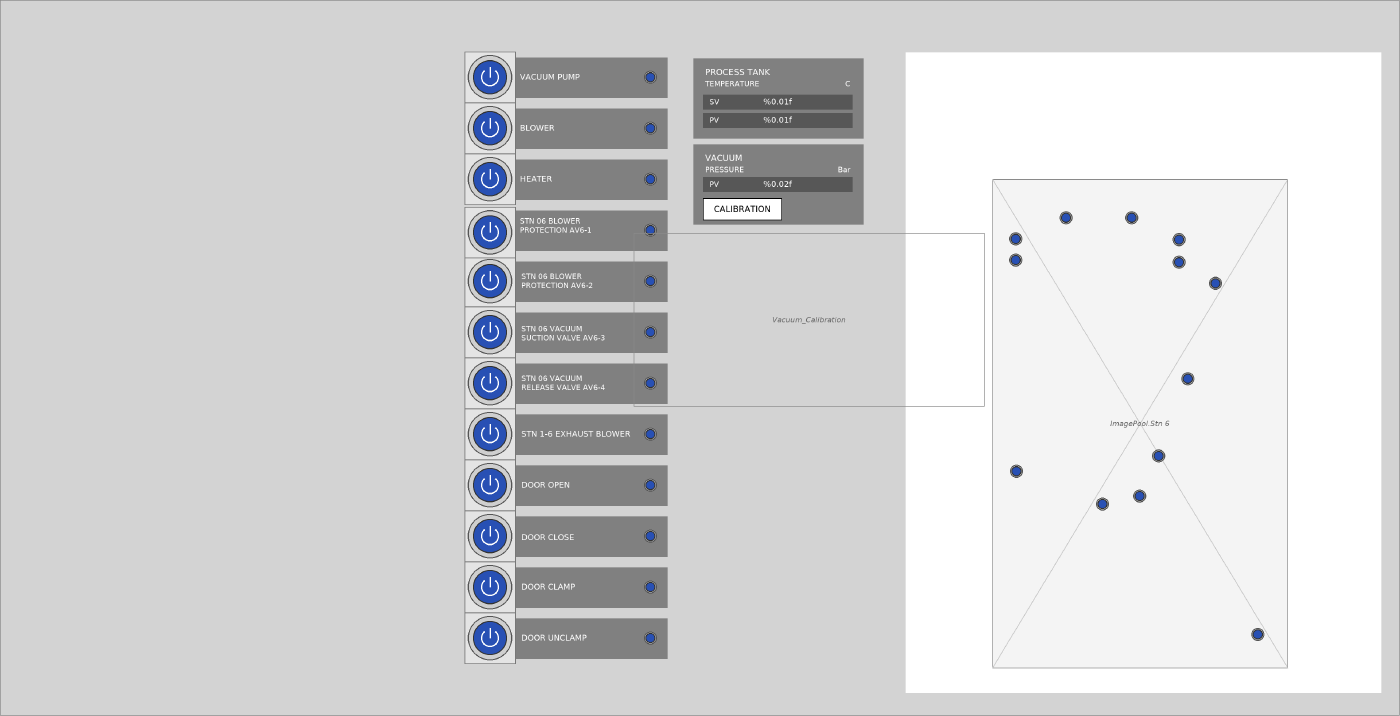
VISUALIZATION Manual_Station06  // 1920x983
    Rectangle (0,0 1920x983)
    Rectangle (1242,72 652x879)
    Image (1361,246 405x671), image: ImagePool.Stn 6
    RoundedRectangle (676,79 239x55)
    Label (710,98 163x16), "VACUUM PUMP"
    Lamp1 (882,96 20x20), variable: ARdsMAP_HmiVariableStn[6].bProTankVacuumPump_IND, style: Lamp-Lamp1-Blue
    PowerSwitch (637,71 70x70), variable: ARdsMAP_HmiVariableStn[6].bProTankVacuumPump_PB, behaviour: TOGGLE, style: Switch-PowerSwitch-Blue
    RoundedRectangle (684,149 231x55)
    Label (710,168 151x16), "BLOWER"
    Lamp1 (882,166 20x20), variable: ARdsMAP_HmiVariableStn[6].bProTankBlower_IND, style: Lamp-Lamp1-Blue
    PowerSwitch (637,141 70x70), variable: ARdsMAP_HmiVariableStn[6].bProTankBlower_PB, behaviour: TOGGLE, style: Switch-PowerSwitch-Blue
    RoundedRectangle (684,219 231x55)
    Label (710,238 151x16), "HEATER"
    Lamp1 (882,236 20x20), variable: ARdsMAP_HmiVariableStn[6].bProTankHeater_IND, style: Lamp-Lamp1-Blue
    PowerSwitch (637,211 70x70), variable: ARdsMAP_HmiVariableStn[6].bProTankHeater_PB, behaviour: TOGGLE, style: Switch-PowerSwitch-Blue
    RoundedRectangle (951,80 233x110)
    Label (964,91 150x16), "PROCESS TANK"
    Label (964,104 99x22), "TEMPERATURE"
    Label (1140,104 29x22), "C"
    Rectangle (964,130 205x20), "%0.01f", text variable: ARrStnTempSV[6]
    Label (970,129 22x22), "SV"
    Rectangle (964,155 205x20), "%0.01f", text variable: ARrStnTempPV[6]
    Label (970,154 50x22), "PV"
    RoundedRectangle (684,359 231x55)
    Label (712,368 160x36), "STN 06 BLOWER PROTECTION AV6-2"
    Lamp1 (882,376 20x20), variable: ARdsMAP_HmiVariableStn[6].bValve02_IND, style: Lamp-Lamp1-Blue
    PowerSwitch (637,351 70x70), variable: ARdsMAP_HmiVariableStn[6].bValve02_PB, behaviour: TOGGLE, style: Switch-PowerSwitch-Blue
    RoundedRectangle (684,499 231x55)
    Label (712,508 160x36), "STN 06 VACUUM RELEASE VALVE AV6-4"
    Lamp1 (882,516 20x20), variable: ARdsMAP_HmiVariableStn[6].bValve04_IND, style: Lamp-Lamp1-Blue
    PowerSwitch (637,491 70x70), variable: ARdsMAP_HmiVariableStn[6].bValve04_PB, behaviour: TOGGLE, style: Switch-PowerSwitch-Blue
    RoundedRectangle (684,429 231x55)
    Lamp1 (882,446 20x20), variable: ARdsMAP_HmiVariableStn[6].bValve03_IND, style: Lamp-Lamp1-Blue
    PowerSwitch (637,421 70x70), variable: ARdsMAP_HmiVariableStn[6].bValve03_PB, behaviour: TOGGLE, style: Switch-PowerSwitch-Blue
    Label (712,440 151x36), "STN 06 VACUUM SUCTION VALVE AV6-3"
    RoundedRectangle (684,569 231x55)
    Label (712,578 160x36), "STN 1-6 EXHAUST BLOWER"
    Lamp1 (882,586 20x20), variable: ARdsMAP_HmiVariableGeneral.bExhaustBlower_IND, style: Lamp-Lamp1-Blue
    PowerSwitch (637,561 70x70), variable: ARdsMAP_HmiVariableGeneral.bExhaustBlower_PB, behaviour: TOGGLE, style: Switch-PowerSwitch-Blue
    RoundedRectangle (684,289 231x55)
    Label (710,298 160x36), "STN 06 BLOWER PROTECTION AV6-1"
    Lamp1 (882,306 20x20), variable: ARdsMAP_HmiVariableStn[6].bValve01_IND, style: Lamp-Lamp1-Blue
    PowerSwitch (637,284 70x70), variable: ARdsMAP_HmiVariableStn[6].bValve01_PB, behaviour: TOGGLE, style: Switch-PowerSwitch-Blue
    Lamp1 (1715,861 20x20), variable: ARdsMAP_HmiVariableStn[6].bProTankVacuumPump_IND, style: Lamp-Lamp1-Blue
    Lamp1 (1553,671 20x20), variable: ARdsMAP_HmiVariableStn[6].bProTankBlower_IND, style: Lamp-Lamp1-Blue
    Lamp1 (1502,682 20x20), variable: ARdsMAP_HmiVariableStn[6].bProTankHeater_IND, style: Lamp-Lamp1-Blue
    Lamp1 (1579,616 20x20), variable: ARdsMAP_HmiVariableStn[6].bValve02_IND, style: Lamp-Lamp1-Blue
    Lamp1 (1657,379 20x20), variable: ARdsMAP_HmiVariableStn[6].bValve04_IND, style: Lamp-Lamp1-Blue
    Lamp1 (1619,510 20x20), variable: ARdsMAP_HmiVariableStn[6].bValve03_IND, style: Lamp-Lamp1-Blue
    Lamp1 (1384,637 20x20), variable: ARdsMAP_HmiVariableStn[6].bValve01_IND, style: Lamp-Lamp1-Blue
    RoundedRectangle (684,639 231x55)
    Label (712,648 160x36), "DOOR OPEN"
    Lamp1 (882,656 20x20), variable: ARbDO[eY12200_Stn06SlidingDoor_Open], style: Lamp-Lamp1-Blue
    PowerSwitch (637,631 70x70), variable: ARwDO[eY12200_Stn06SlidingDoor_Open].15, behaviour: TOGGLE, style: Switch-PowerSwitch-Blue
    RoundedRectangle (684,779 231x55)
    Label (712,788 160x36), "DOOR CLAMP"
    Lamp1 (882,796 20x20), variable: ARbDO[eY12202_Stn06SlidingDoor_Clamp], style: Lamp-Lamp1-Blue
    PowerSwitch (637,771 70x70), variable: ARwDO[eY12202_Stn06SlidingDoor_Clamp].15, behaviour: TOGGLE, style: Switch-PowerSwitch-Blue
    RoundedRectangle (684,709 231x55)
    Lamp1 (882,726 20x20), variable: ARbDO[eY12201_Stn06SlidingDoor_Close], style: Lamp-Lamp1-Blue
    PowerSwitch (637,701 70x70), variable: ARwDO[eY12201_Stn06SlidingDoor_Close].15, behaviour: TOGGLE, style: Switch-PowerSwitch-Blue
    Label (712,720 151x36), "DOOR CLOSE"
    RoundedRectangle (684,849 231x55)
    Label (712,858 160x36), "DOOR UNCLAMP"
    PowerSwitch (637,841 70x70), variable: ARwDO[eY12203_Stn06SlidingDoor_Unclamp].15, behaviour: TOGGLE, style: Switch-PowerSwitch-Blue
    Lamp1 (882,866 20x20), variable: ARbDO[eY12203_Stn06SlidingDoor_Unclamp], style: Lamp-Lamp1-Blue
    Lamp1 (1383,347 20x20), variable: ARbDI[eX12100_Stn06SlidingDoorRs01_Clamp], style: Lamp-Lamp1-Blue
    Lamp1 (1607,350 20x20), variable: ARbDI[eX12102_Stn06SlidingDoorRs02_Clamp], style: Lamp-Lamp1-Blue
    Lamp1 (1383,318 20x20), variable: ARbDI[eX12101_Stn06SlidingDoorRs01_Unclamp], style: Lamp-Lamp1-Blue
    Lamp1 (1607,319 20x20), variable: ARbDI[eX12103_Stn06SlidingDoorRs02_Unclamp], style: Lamp-Lamp1-Blue
    Lamp1 (1542,289 20x20), variable: ARbDI[eX12008_Stn06SlidingDoorRs_Close], style: Lamp-Lamp1-Blue
    Lamp1 (1452,289 20x20), variable: ARbDI[eX12007_Stn06SlidingDoorRs_Open], style: Lamp-Lamp1-Blue
    RoundedRectangle (951,198 233x110)
    Label (964,209 150x16), "VACUUM"
    Label (964,222 99x22), "PRESSURE"
    Label (1145,222 24x22), "Bar"
    Rectangle (964,243 205x20), "%0.02f", text variable: ARrStnVacuumPV[6]
    Label (970,242 57x22), "PV"
    Rectangle (964,272 108x30), "CALIBRATION", colour toggle: ARDSProminentDosingHMI[iSettingStnNo].In_bResetRemainedDosingVolumePB
        tap ARDSProminentDosingHMI[HMI_Ctrl.StationInfoPageNo].In_bResetRemainedDosingVolumePB
        toggle bManualCalibratePageOn
    Frame (869,320 481x238), invisible if: bManualCalibratePageOn
        shows Vacuum_Calibration()
END_VISUALIZATION

(* stored: Version 1.1.0.1, ProductVersion 3.1.4024.12
   Visu Manual_Station06: Id {bf90e307-f400-4e99-b447-e29ad010f0d3} *)
